{attribute 'GeneratedUsingTerminal: KL2012'}
{attribute addProperty BoxType "KL2012"}
{attribute addProperty Id "OutputAT %Q*BOOL0"}
{attribute addProperty CRC "1175161920"}
{attribute addProperty Size "0"}
TYPE Channel_460B8C40 :
STRUCT
	{attribute addProperty Name "Output"}
	Output AT %Q* : BOOL;
END_STRUCT
END_TYPE

(* stored: Version 1.2.0.0, ProductVersion 3.1.4024.9
   DUT Channel_460B8C40: Id {7b8d8a52-ae3c-4f8a-9fcb-cdc81626f35c} *)
